SYSTEM test_PUBLISH_SUBSCRIBE
  (* Version 1.0, 2023-10-23, Franz Höpfinger, Meisterschulen am Ostbahnhof *)
  PACKAGE Training_PUBLISH_SUBSCRIBE;
  IMPORT logiBUS::io::DI::logiBUS_DI::Input_I1;
  IMPORT logiBUS::io::DI::logiBUS_DI::Input_I2;
  IMPORT logiBUS::io::DI::logiBUS_DI::Input_I3;
  IMPORT logiBUS::io::DI::logiBUS_DI::Input_I4;
  IMPORT logiBUS::io::DO_LED::LED_COLOURS::LED_BLUE;
  IMPORT logiBUS::io::DO_LED::LED_COLOURS::LED_GREEN;
  IMPORT logiBUS::io::DO_LED::LED_COLOURS::LED_RED;
  IMPORT logiBUS::io::DO_LED::LED_COLOURS::LED_YELLOW;
  IMPORT logiBUS::io::DO_LED::LED_FREQ::LED_5HZ;
  IMPORT logiBUS::io::DO_LED::LED_strip::Output_strip;
  APPLICATION App_PUBLISH_SUBSCRIBE
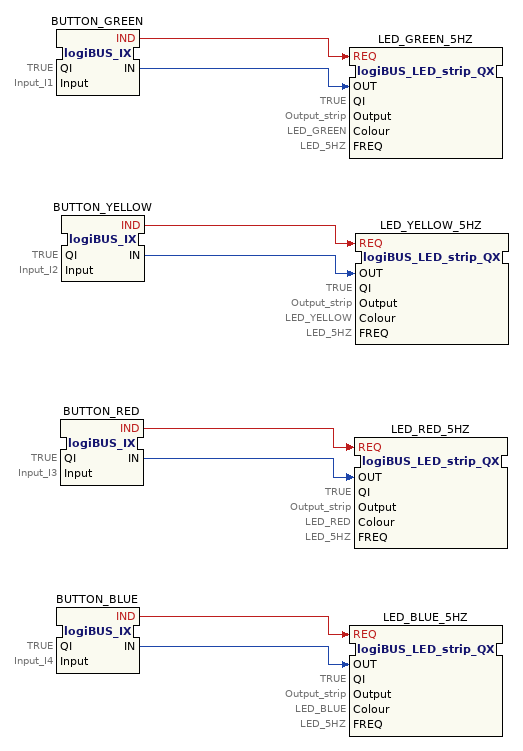
    FBS
      BUTTON_RED : logiBUS::io::DI::logiBUS_IX(QI := TRUE, Input := Input_I3);
      BUTTON_YELLOW : logiBUS::io::DI::logiBUS_IX(QI := TRUE, Input := Input_I2);
      BUTTON_BLUE : logiBUS::io::DI::logiBUS_IX(QI := TRUE, Input := Input_I4);
      LED_YELLOW_5HZ : logiBUS::io::DO_LED::logiBUS_LED_strip_QX(QI := TRUE, Output := Output_strip, Colour := LED_YELLOW, FREQ := LED_5HZ);
      LED_BLUE_5HZ : logiBUS::io::DO_LED::logiBUS_LED_strip_QX(QI := TRUE, Output := Output_strip, Colour := LED_BLUE, FREQ := LED_5HZ);
      LED_RED_5HZ : logiBUS::io::DO_LED::logiBUS_LED_strip_QX(QI := TRUE, Output := Output_strip, Colour := LED_RED, FREQ := LED_5HZ);
      BUTTON_GREEN : logiBUS::io::DI::logiBUS_IX(QI := TRUE, Input := Input_I1);
      LED_GREEN_5HZ : logiBUS::io::DO_LED::logiBUS_LED_strip_QX(QI := TRUE, Output := Output_strip, Colour := LED_GREEN, FREQ := LED_5HZ);
    END_FBS
    EVENT_CONNECTIONS
      BUTTON_RED.IND TO LED_RED_5HZ.REQ;
      BUTTON_YELLOW.IND TO LED_YELLOW_5HZ.REQ;
      BUTTON_BLUE.IND TO LED_BLUE_5HZ.REQ;
      BUTTON_GREEN.IND TO LED_GREEN_5HZ.REQ;
    END_CONNECTIONS
    DATA_CONNECTIONS
      BUTTON_RED.IN TO LED_RED_5HZ.OUT;
      BUTTON_YELLOW.IN TO LED_YELLOW_5HZ.OUT;
      BUTTON_BLUE.IN TO LED_BLUE_5HZ.OUT;
      BUTTON_GREEN.IN TO LED_GREEN_5HZ.OUT;
    END_CONNECTIONS
  END_APPLICATION
  DEVICE FORTE_PC_PUBLISH : iec61499::system::FORTE_PC(MGR_ID := VV::const::Computers::myComputers::C_PC_PUBLISH (* Device manager socket ID *))
    {SET_ATTRIBUTE(Profile, OPC UA)}
    RESOURCE EMB_RES_PUBLISH : iec61499::system::EMB_RES
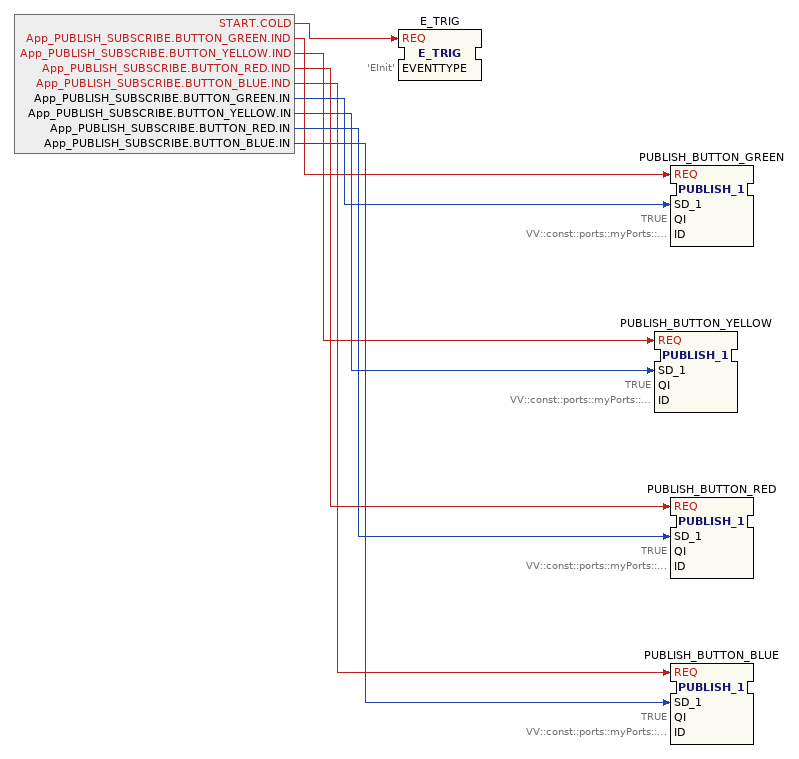
      FBS
        PUBLISH_BUTTON_GREEN : iec61499::net::PUBLISH_1(QI := TRUE, ID := VV::const::ports::myPorts::PORT_0);
        PUBLISH_BUTTON_YELLOW : iec61499::net::PUBLISH_1(QI := TRUE, ID := VV::const::ports::myPorts::PORT_1);
        PUBLISH_BUTTON_RED : iec61499::net::PUBLISH_1(QI := TRUE, ID := VV::const::ports::myPorts::PORT_2);
        PUBLISH_BUTTON_BLUE : iec61499::net::PUBLISH_1(QI := TRUE, ID := VV::const::ports::myPorts::PORT_3);
        E_TRIG : iec61499::events::E_TRIG(EVENTTYPE := 'EInit');
      END_FBS
      EVENT_CONNECTIONS
        START.COLD TO E_TRIG.REQ;
        App_PUBLISH_SUBSCRIBE.BUTTON_GREEN.IND TO PUBLISH_BUTTON_GREEN.REQ;
        App_PUBLISH_SUBSCRIBE.BUTTON_YELLOW.IND TO PUBLISH_BUTTON_YELLOW.REQ;
        App_PUBLISH_SUBSCRIBE.BUTTON_RED.IND TO PUBLISH_BUTTON_RED.REQ;
        App_PUBLISH_SUBSCRIBE.BUTTON_BLUE.IND TO PUBLISH_BUTTON_BLUE.REQ;
      END_CONNECTIONS
      DATA_CONNECTIONS
        App_PUBLISH_SUBSCRIBE.BUTTON_GREEN.IN TO PUBLISH_BUTTON_GREEN.SD_1;
        App_PUBLISH_SUBSCRIBE.BUTTON_YELLOW.IN TO PUBLISH_BUTTON_YELLOW.SD_1;
        App_PUBLISH_SUBSCRIBE.BUTTON_RED.IN TO PUBLISH_BUTTON_RED.SD_1;
        App_PUBLISH_SUBSCRIBE.BUTTON_BLUE.IN TO PUBLISH_BUTTON_BLUE.SD_1;
      END_CONNECTIONS
    END_RESOURCE
  END_DEVICE
  DEVICE FORTE_PC_SUBSCRIBE : iec61499::system::FORTE_PC(MGR_ID := VV::const::Computers::myComputers::C_PC_SUBSCRIBE (* Device manager socket ID *))
    {SET_ATTRIBUTE(Profile, OPC UA)}
    RESOURCE EMB_RES_SUBSCRIBE : iec61499::system::EMB_RES
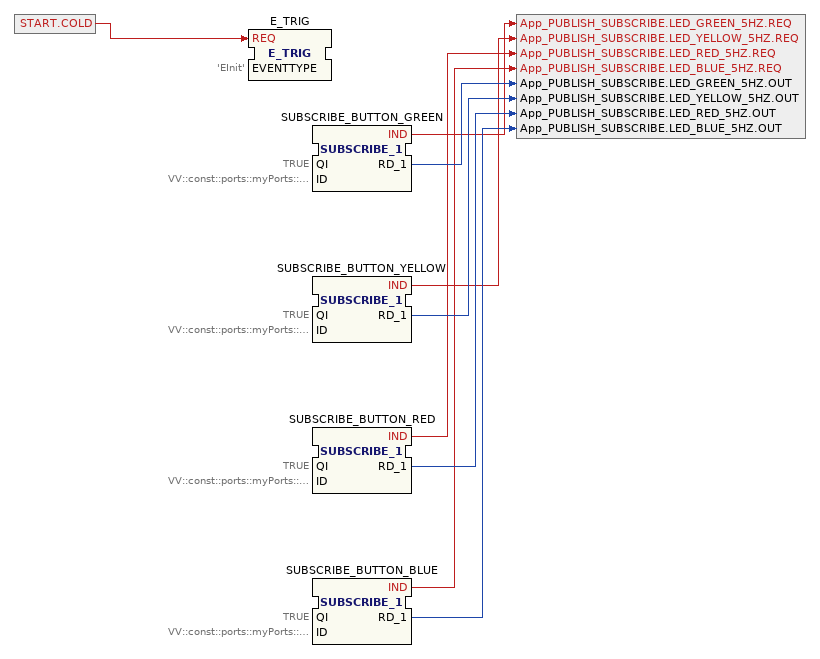
      FBS
        SUBSCRIBE_BUTTON_GREEN : iec61499::net::SUBSCRIBE_1(QI := TRUE, ID := VV::const::ports::myPorts::PORT_0);
        SUBSCRIBE_BUTTON_YELLOW : iec61499::net::SUBSCRIBE_1(QI := TRUE, ID := VV::const::ports::myPorts::PORT_1);
        SUBSCRIBE_BUTTON_RED : iec61499::net::SUBSCRIBE_1(QI := TRUE, ID := VV::const::ports::myPorts::PORT_2);
        SUBSCRIBE_BUTTON_BLUE : iec61499::net::SUBSCRIBE_1(QI := TRUE, ID := VV::const::ports::myPorts::PORT_3);
        E_TRIG : iec61499::events::E_TRIG(EVENTTYPE := 'EInit');
      END_FBS
      EVENT_CONNECTIONS
        START.COLD TO E_TRIG.REQ;
        SUBSCRIBE_BUTTON_GREEN.IND TO App_PUBLISH_SUBSCRIBE.LED_GREEN_5HZ.REQ;
        SUBSCRIBE_BUTTON_YELLOW.IND TO App_PUBLISH_SUBSCRIBE.LED_YELLOW_5HZ.REQ;
        SUBSCRIBE_BUTTON_RED.IND TO App_PUBLISH_SUBSCRIBE.LED_RED_5HZ.REQ;
        SUBSCRIBE_BUTTON_BLUE.IND TO App_PUBLISH_SUBSCRIBE.LED_BLUE_5HZ.REQ;
      END_CONNECTIONS
      DATA_CONNECTIONS
        SUBSCRIBE_BUTTON_GREEN.RD_1 TO App_PUBLISH_SUBSCRIBE.LED_GREEN_5HZ.OUT;
        SUBSCRIBE_BUTTON_YELLOW.RD_1 TO App_PUBLISH_SUBSCRIBE.LED_YELLOW_5HZ.OUT;
        SUBSCRIBE_BUTTON_RED.RD_1 TO App_PUBLISH_SUBSCRIBE.LED_RED_5HZ.OUT;
        SUBSCRIBE_BUTTON_BLUE.RD_1 TO App_PUBLISH_SUBSCRIBE.LED_BLUE_5HZ.OUT;
      END_CONNECTIONS
    END_RESOURCE
  END_DEVICE
  MAPPINGS
    App_PUBLISH_SUBSCRIBE.BUTTON_BLUE ON FORTE_PC_PUBLISH.EMB_RES_PUBLISH;
    App_PUBLISH_SUBSCRIBE.BUTTON_RED ON FORTE_PC_PUBLISH.EMB_RES_PUBLISH;
    App_PUBLISH_SUBSCRIBE.BUTTON_YELLOW ON FORTE_PC_PUBLISH.EMB_RES_PUBLISH;
    App_PUBLISH_SUBSCRIBE.LED_RED_5HZ ON FORTE_PC_SUBSCRIBE.EMB_RES_SUBSCRIBE;
    App_PUBLISH_SUBSCRIBE.LED_YELLOW_5HZ ON FORTE_PC_SUBSCRIBE.EMB_RES_SUBSCRIBE;
    App_PUBLISH_SUBSCRIBE.LED_BLUE_5HZ ON FORTE_PC_SUBSCRIBE.EMB_RES_SUBSCRIBE;
    App_PUBLISH_SUBSCRIBE.LED_GREEN_5HZ ON FORTE_PC_SUBSCRIBE.EMB_RES_SUBSCRIBE;
    App_PUBLISH_SUBSCRIBE.BUTTON_GREEN ON FORTE_PC_PUBLISH.EMB_RES_PUBLISH;
  END_MAPPINGS
  SEGMENTS
    Ethernet : iec61499::system::Ethernet;
  END_SEGMENTS
  LINKS
    FORTE_PC_PUBLISH => Ethernet;
    FORTE_PC_SUBSCRIBE => Ethernet;
  END_LINKS
END_SYSTEM
